FUNCTION_BLOCK Conveyor_View_Small (* Composite Function Block Type *)
  (* Standard: 61499-2 *)
  (* Version 0.2, 2003-12-05, JHC, Rockwell Automation, Renamed from NEWCOMPFB. *)
  (* Version 0.1, 2002-01-08, JHC, Rockwell Automation, Added DLY FB as example. *)
  (* Version 0.0, 2000-05-27, JHC, Rockwell Automation *)
  (* Compiler header: package fb.rt.cs725;import fb.rt.vhmi.*; *)
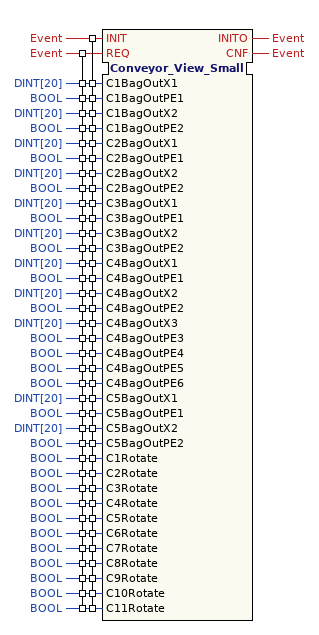
  EVENT_INPUT
    INIT WITH C1BagOutX1, C1BagOutPE1, C1BagOutX2, C1BagOutPE2, C2BagOutX1, C2BagOutPE1, C2BagOutX2, C2BagOutPE2, C3BagOutX1, C3BagOutPE1, C3BagOutX2, C3BagOutPE2, C4BagOutX1, C4BagOutPE1, C4BagOutX2, C4BagOutPE2, C4BagOutX3, C4BagOutPE3, C4BagOutPE4, C4BagOutPE5, C1Rotate, C2Rotate, C3Rotate, C4Rotate, C5Rotate, C6Rotate, C7Rotate, C8Rotate, C9Rotate, C10Rotate, C11Rotate, C4BagOutPE6, C5BagOutX1, C5BagOutPE1, C5BagOutX2, C5BagOutPE2; (* Initialization Request *)
    REQ WITH C1BagOutX1, C1BagOutPE1, C1BagOutX2, C1BagOutPE2, C2BagOutX1, C2BagOutPE1, C2BagOutX2, C2BagOutPE2, C3BagOutX1, C3BagOutPE1, C3BagOutX2, C3BagOutPE2, C4BagOutX1, C4BagOutPE1, C4BagOutX2, C4BagOutPE2, C4BagOutX3, C4BagOutPE3, C4BagOutPE4, C4BagOutPE5, C1Rotate, C2Rotate, C3Rotate, C4Rotate, C5Rotate, C6Rotate, C7Rotate, C8Rotate, C9Rotate, C10Rotate, C11Rotate, C4BagOutPE6, C5BagOutX1, C5BagOutPE1, C5BagOutX2, C5BagOutPE2; (* Normal Execution Request *)
  END_EVENT
  EVENT_OUTPUT
    INITO; (* Initialization Confirm *)
    CNF; (* Execution Confirmation *)
  END_EVENT
  VAR_INPUT
    C1BagOutX1 : ARRAY [0..19] OF DINT;
    C1BagOutPE1 : BOOL;
    C1BagOutX2 : ARRAY [0..19] OF DINT;
    C1BagOutPE2 : BOOL;
    C2BagOutX1 : ARRAY [0..19] OF DINT;
    C2BagOutPE1 : BOOL;
    C2BagOutX2 : ARRAY [0..19] OF DINT;
    C2BagOutPE2 : BOOL;
    C3BagOutX1 : ARRAY [0..19] OF DINT;
    C3BagOutPE1 : BOOL;
    C3BagOutX2 : ARRAY [0..19] OF DINT;
    C3BagOutPE2 : BOOL;
    C4BagOutX1 : ARRAY [0..19] OF DINT;
    C4BagOutPE1 : BOOL;
    C4BagOutX2 : ARRAY [0..19] OF DINT;
    C4BagOutPE2 : BOOL;
    C4BagOutX3 : ARRAY [0..19] OF DINT;
    C4BagOutPE3 : BOOL;
    C4BagOutPE4 : BOOL;
    C4BagOutPE5 : BOOL;
    C4BagOutPE6 : BOOL;
    C5BagOutX1 : ARRAY [0..19] OF DINT;
    C5BagOutPE1 : BOOL;
    C5BagOutX2 : ARRAY [0..19] OF DINT;
    C5BagOutPE2 : BOOL;
    C1Rotate : BOOL;
    C2Rotate : BOOL;
    C3Rotate : BOOL;
    C4Rotate : BOOL;
    C5Rotate : BOOL;
    C6Rotate : BOOL;
    C7Rotate : BOOL;
    C8Rotate : BOOL;
    C9Rotate : BOOL;
    C10Rotate : BOOL;
    C11Rotate : BOOL;
  END_VAR
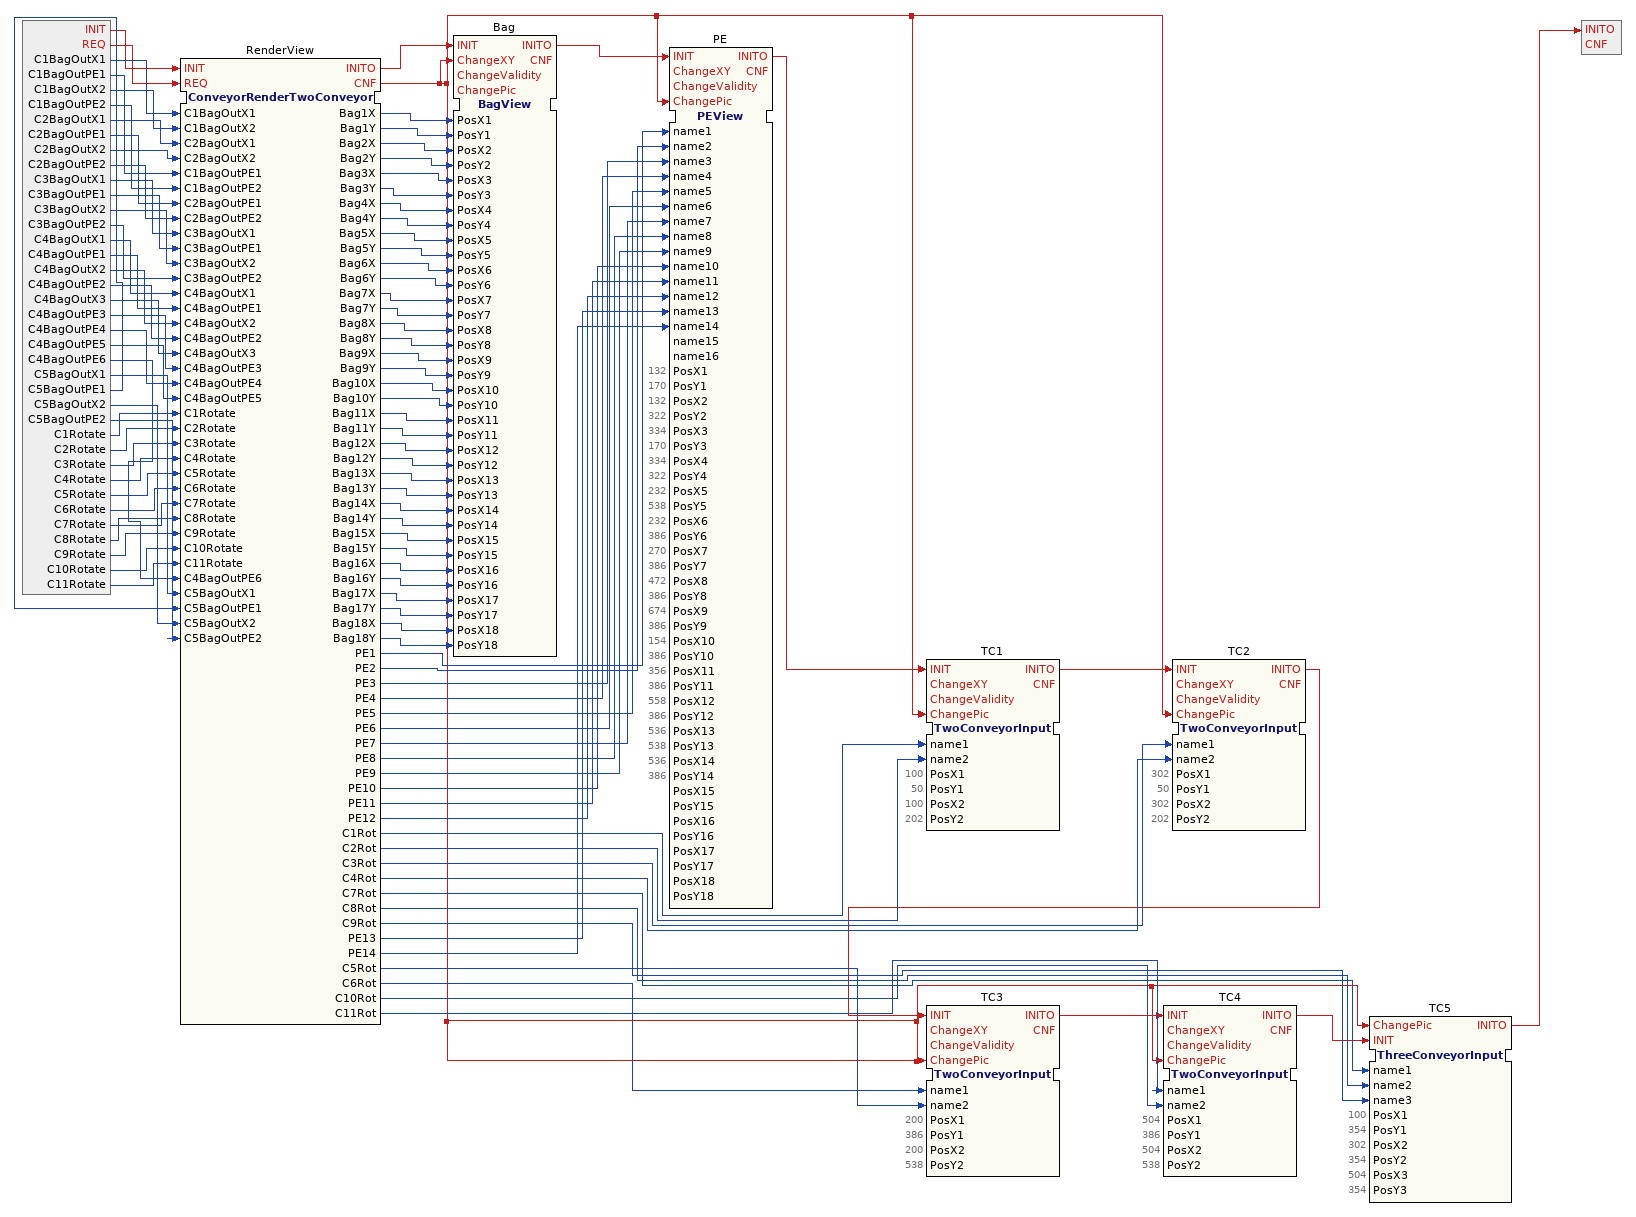
  FBS
    RenderView : ConveyorRenderTwoConveyor;
    Bag : BagView;
    PE : PEView(PosX1 := 132, PosX2 := 132, PosY1 := 170, PosY2 := 322, PosX3 := 334, PosX4 := 334, PosY3 := 170, PosY4 := 322, PosX5 := 232, PosX6 := 232, PosY5 := 538, PosY6 := 386, PosX7 := 270, PosY7 := 386, PosY8 := 386, PosY9 := 386, PosX8 := 472, PosX9 := 674, PosX10 := 154, PosY10 := 386, PosX11 := 356, PosY11 := 386, PosX13 := 536, PosY13 := 538, PosX14 := 536, PosY14 := 386, PosX12 := 558, PosY12 := 386);
    TC1 : TwoConveyorInput(PosX1 := 100, PosY1 := 50, PosX2 := 100, PosY2 := 202);
    TC2 : TwoConveyorInput(PosX1 := 302, PosY1 := 50, PosX2 := 302, PosY2 := 202);
    TC3 : TwoConveyorInput(PosX1 := 200, PosY1 := 386, PosX2 := 200, PosY2 := 538);
    TC5 : ThreeConveyorInput(PosX1 := 100, PosY1 := 354, PosX2 := 302, PosY2 := 354, PosX3 := 504, PosY3 := 354);
    TC4 : TwoConveyorInput(PosX1 := 504, PosY1 := 386, PosX2 := 504, PosY2 := 538);
  END_FBS
  EVENT_CONNECTIONS
    INIT TO RenderView.INIT;
    REQ TO RenderView.REQ;
    RenderView.INITO TO Bag.INIT;
    RenderView.CNF TO Bag.ChangeXY;
    Bag.INITO TO PE.INIT;
    RenderView.CNF TO PE.ChangePic;
    PE.INITO TO TC1.INIT;
    TC1.INITO TO TC2.INIT;
    TC2.INITO TO TC3.INIT;
    TC5.INITO TO INITO;
    RenderView.CNF TO TC1.ChangePic;
    RenderView.CNF TO TC2.ChangePic;
    RenderView.CNF TO TC3.ChangePic;
    RenderView.CNF TO TC5.ChangePic;
    TC3.INITO TO TC4.INIT;
    TC4.INITO TO TC5.INIT;
    RenderView.CNF TO TC4.ChangePic;
  END_CONNECTIONS
  DATA_CONNECTIONS
    RenderView.Bag1X TO Bag.PosX1;
    RenderView.Bag1Y TO Bag.PosY1;
    RenderView.Bag2X TO Bag.PosX2;
    RenderView.Bag2Y TO Bag.PosY2;
    RenderView.Bag3X TO Bag.PosX3;
    RenderView.Bag3Y TO Bag.PosY3;
    RenderView.Bag4X TO Bag.PosX4;
    RenderView.Bag4Y TO Bag.PosY4;
    RenderView.Bag5X TO Bag.PosX5;
    RenderView.Bag5Y TO Bag.PosY5;
    RenderView.Bag6X TO Bag.PosX6;
    RenderView.Bag6Y TO Bag.PosY6;
    RenderView.Bag7X TO Bag.PosX7;
    RenderView.Bag7Y TO Bag.PosY7;
    RenderView.Bag8X TO Bag.PosX8;
    RenderView.Bag8Y TO Bag.PosY8;
    RenderView.Bag9X TO Bag.PosX9;
    RenderView.Bag9Y TO Bag.PosY9;
    RenderView.Bag10X TO Bag.PosX10;
    RenderView.Bag10Y TO Bag.PosY10;
    RenderView.Bag11X TO Bag.PosX11;
    RenderView.Bag11Y TO Bag.PosY11;
    RenderView.Bag12X TO Bag.PosX12;
    RenderView.Bag12Y TO Bag.PosY12;
    RenderView.Bag13X TO Bag.PosX13;
    RenderView.Bag13Y TO Bag.PosY13;
    RenderView.Bag14X TO Bag.PosX14;
    RenderView.Bag14Y TO Bag.PosY14;
    RenderView.Bag15X TO Bag.PosX15;
    RenderView.Bag15Y TO Bag.PosY15;
    RenderView.Bag16X TO Bag.PosX16;
    RenderView.Bag16Y TO Bag.PosY16;
    RenderView.Bag17X TO Bag.PosX17;
    RenderView.Bag17Y TO Bag.PosY17;
    RenderView.Bag18X TO Bag.PosX18;
    RenderView.Bag18Y TO Bag.PosY18;
    C1BagOutX1 TO RenderView.C1BagOutX1;
    C1BagOutX2 TO RenderView.C1BagOutX2;
    C2BagOutX1 TO RenderView.C2BagOutX1;
    C2BagOutX2 TO RenderView.C2BagOutX2;
    C1BagOutPE1 TO RenderView.C1BagOutPE1;
    C1BagOutPE2 TO RenderView.C1BagOutPE2;
    C2BagOutPE1 TO RenderView.C2BagOutPE1;
    C2BagOutPE2 TO RenderView.C2BagOutPE2;
    C3BagOutX1 TO RenderView.C3BagOutX1;
    C3BagOutPE1 TO RenderView.C3BagOutPE1;
    C3BagOutX2 TO RenderView.C3BagOutX2;
    C3BagOutPE2 TO RenderView.C3BagOutPE2;
    C4BagOutX1 TO RenderView.C4BagOutX1;
    C4BagOutPE1 TO RenderView.C4BagOutPE1;
    C4BagOutX2 TO RenderView.C4BagOutX2;
    C4BagOutPE2 TO RenderView.C4BagOutPE2;
    C4BagOutX3 TO RenderView.C4BagOutX3;
    C4BagOutPE3 TO RenderView.C4BagOutPE3;
    RenderView.PE1 TO PE.name1;
    RenderView.PE2 TO PE.name2;
    RenderView.PE3 TO PE.name3;
    RenderView.PE4 TO PE.name4;
    RenderView.PE5 TO PE.name5;
    RenderView.PE6 TO PE.name6;
    RenderView.PE7 TO PE.name7;
    RenderView.PE8 TO PE.name8;
    RenderView.PE9 TO PE.name9;
    RenderView.PE10 TO PE.name10;
    RenderView.PE11 TO PE.name11;
    RenderView.PE12 TO PE.name12;
    C4BagOutPE4 TO RenderView.C4BagOutPE4;
    C4BagOutPE5 TO RenderView.C4BagOutPE5;
    RenderView.C1Rot TO TC1.name1;
    RenderView.C2Rot TO TC1.name2;
    RenderView.C3Rot TO TC2.name1;
    RenderView.C4Rot TO TC2.name2;
    RenderView.C7Rot TO TC5.name1;
    RenderView.C8Rot TO TC5.name2;
    RenderView.C9Rot TO TC5.name3;
    C1Rotate TO RenderView.C1Rotate;
    C2Rotate TO RenderView.C2Rotate;
    C3Rotate TO RenderView.C3Rotate;
    C4Rotate TO RenderView.C4Rotate;
    C5Rotate TO RenderView.C5Rotate;
    C6Rotate TO RenderView.C6Rotate;
    C7Rotate TO RenderView.C7Rotate;
    C8Rotate TO RenderView.C8Rotate;
    C9Rotate TO RenderView.C9Rotate;
    RenderView.PE13 TO PE.name13;
    RenderView.PE14 TO PE.name14;
    C10Rotate TO RenderView.C10Rotate;
    C11Rotate TO RenderView.C11Rotate;
    C4BagOutPE6 TO RenderView.C4BagOutPE6;
    C5BagOutX1 TO RenderView.C5BagOutX1;
    C5BagOutPE1 TO RenderView.C5BagOutPE1;
    C5BagOutX2 TO RenderView.C5BagOutX2;
    C5BagOutPE2 TO RenderView.C5BagOutPE2;
    RenderView.C5Rot TO TC3.name2;
    RenderView.C6Rot TO TC3.name1;
    RenderView.C10Rot TO TC4.name2;
    RenderView.C11Rot TO TC4.name1;
  END_CONNECTIONS
END_FUNCTION_BLOCK
